FUNCTION_BLOCK GreenMasterBaseParametersFB
VAR_IN_OUT
	GreenMaster: GreenMasterBase;
END_VAR
VAR_INPUT
END_VAR
VAR_OUTPUT
	System: SystemParametersFB;
	Regulation: RegulationParametersFB;
	//Alarm: AlarmParametersFB;
	IO: IoParametersFB;
	Simulation: SimulationFB;
END_VAR
VAR
END_VAR

System(ParametersFB := THIS^, Parameters := GreenMaster.GetParameters(), System := GreenMaster.GetParameters().System);
Regulation(ParametersFB := THIS^, Parameters := GreenMaster.GetParameters(), Regulation := GreenMaster.GetParameters().Regulation);
IO(GreenMaster := GreenMaster, ParametersFB := THIS^, Parameters := GreenMaster.GetParameters());

METHOD GetGreenMaster : REFERENCE TO GreenMasterBase
VAR_INPUT
END_VAR
GetGreenMaster REF= GreenMaster;
END_METHOD

END_FUNCTION_BLOCK

(* stored: Version 1.1.0.1, ProductVersion 3.1.4024.6
   POU GreenMasterBaseParametersFB: Id {4f104a97-9854-4cb1-aeb3-f00bd259eb43}, SpecialFunc None
   Method GetGreenMaster: Id {8a59516c-2d19-481f-8e6e-4d8f0472c8c1} *)
